FUNCTION AxesMoveUnitsToDeg : LREAL
VAR_INPUT
    units : AxesMoveUnits;
    value : LREAL;
END_VAR
VAR
END_VAR

CASE units OF
    AxesMoveUnits.RADIANS:
        AxesMoveUnitsToDeg := RAD_TO_DEG(value);
    AxesMoveUnits.DEGREES:
        AxesMoveUnitsToDeg := value; 
    AxesMoveUnits.ARCSECONDS:
        AxesMoveUnitsToDeg := ARCSEC_TO_DEG(value);   
END_CASE

END_FUNCTION

(* stored: Version 1.1.0.1, ProductVersion 3.1.4018.5
   POU AxesMoveUnitsToDeg: Id {4d77c3eb-6f54-48a7-a6da-2368cb679121}, SpecialFunc None *)
